// TIA Portal V16 export
// export: Created 2023-08-28T09:37:53.340562Z, ExportSetting WithDefaults, DisplayName Totally Integrated Automation Portal, DisplayVersion V16 Update 6, DisplayName TIA Portal Version Control Interface, DisplayVersion V16 Update 2, DisplayName TIA Portal Openness, DisplayVersion V16 Update 6, DisplayName STEP 7 Professional, DisplayVersion V16 Update 6, DisplayName STEP 7 Safety, DisplayVersion V16, DisplayName WinCC Advanced, DisplayVersion V16 Update 6
DATA_BLOCK "01_E_cleaning_the_alarm_reset_button_DB"   // DB48
AUTHOR : rtecme
VERSION : 0.1
// stored: AutoNumber true, DBAccessibleFromOPCUA true, InstanceOfName 01_E_cleaning_the_alarm_reset_button, InstanceOfType FB
"01_E_cleaning_the_alarm_reset_button"
BEGIN
END_DATA_BLOCK
